Fanuc TP program (LS listing): TEST.LS

/PROG  TEST
/ATTR
OWNER		= MNEDITOR;
COMMENT		= "";
PROG_SIZE	= 603;
CREATE		= DATE 23-10-26  TIME 09:44:02;
MODIFIED	= DATE 23-10-26  TIME 09:54:48;
FILE_NAME	= ;
VERSION		= 0;
LINE_COUNT	= 6;
MEMORY_SIZE	= 951;
PROTECT		= READ_WRITE;
TCD:  STACK_SIZE	= 0,
      TASK_PRIORITY	= 50,
      TIME_SLICE	= 0,
      BUSY_LAMP_OFF	= 0,
      ABORT_REQUEST	= 0,
      PAUSE_REQUEST	= 0;
DEFAULT_GROUP	= 1,*,*,*,*;
CONTROL_CODE	= 00000000 00000000;
LOCAL_REGISTERS	= 0,0,0;
/APPL
/APPL

AUTO_SINGULARITY_HEADER;
  ENABLE_SINGULARITY_AVOIDANCE   : FALSE;

PLTZ_MODE_HEADER;
 PLTZ_MODE_ENABLE   : FALSE;
 J4TURN  : ZERORAD;
 ORIENT  : DOWNWARDS;
/MN
   1:  FOR R[35:i]=1 TO 55 ;
   2:  PR[41,3:layer_offset]=213.2*R[35:i]    ;
   3:J P[1] 100% CNT100 Offset,PR[41:layer_offset]    ;
   4:  PAUSE ;
   5:  ENDFOR ;
   6:J P[1] 100% CNT100    ;
/POS
P[1]{
   GP1:
	UF : 1, UT : 9,		CONFIG : 'N U T, 0, 0, 0',
	X =   643.849182  mm,	Y =  1128.170410  mm,	Z =   685.000305  mm,
	W =      .001806 deg,	P =     -.001516 deg,	R =     1.998051 deg
};
/END
